TYPE ST_DB_OACCheckCtrl :
STRUCT
	bDB_ExecuteOacCheck			: BOOL;
	bDB_OacCheckComplete			: BOOL;
	bOacValid						: BOOL;
	bDB_Error						: BOOL;
	stOacToCheck					: ST_OUTER_Status;
END_STRUCT
END_TYPE

(* stored: Version 1.1.0.1, ProductVersion 3.1.4024.15
   DUT ST_DB_OACCheckCtrl: Id {5c5dcd82-396c-49c0-ae41-72b3eef996af} *)
